Fanuc TP program (LS listing): mv_to_pick.ls

/PROG  MV_TO_PICK
/ATTR
DEFAULT_GROUP	= 1,*,*,*,*;
/MN
 : CALL MV_RETREAT ;
 :  ;
 : UFRAME_NUM=${UF_PICK} ;
 : UTOOL_NUM=${UT_PICK} ;
 : J PR{PICK_PERCH} ${PERCH_SPEED}% CNT100 ;
/POS
/END
